Fanuc KAREL source: GET_PORT_MOD.kl

PROGRAM T
%NOLOCKGROUP
VAR
 v0 : INTEGER
 v1 : INTEGER
 v2 : INTEGER
 v3 : INTEGER
BEGIN
 GET_PORT_MOD(v0, v1, v2, v3)
END T
